// TIA Portal V18 export
DATA_BLOCK "Simulation_Data_DB"   // DB1
VERSION : 0.1
// stored: AutoNumber true, DBAccessibleFromOPCUA true, DBAccessibleFromWebserver true, InstanceOfName Simulation_Data, InstanceOfType FB
"Simulation_Data"
   // VAR
   //    Old_Clock : Bool;
   //    i : Int;
   // END_VAR
BEGIN
END_DATA_BLOCK
